TYPE E_ExtruderType :
(
	PistonExtruder1,
	FilamentExtruder1,
	ScrewExtruder1,
	SyringeExtruder1,
	FilamentExtruder2,
	PureDyne_1,
	PureDyne_2,
	PureDyne_3
)USINT;
END_TYPE

(* stored: Version 1.1.0.1
   DUT E_ExtruderType: Id {3e27c3b2-798f-426c-a4fa-288e881d0ab0} *)
